FUNCTION F_ROUNDREAL : REAL
VAR_INPUT
	rValue		: REAL; // Input Value
	iDecNumber	: INT; 	// Numbers after decimal point
END_VAR
VAR
	rOutValue	: REAL;
END_VAR

rOutValue := rValue * EXPT(10,iDecNumber);
rOutValue := TRUNC(rOutValue) / EXPT(10,iDecNumber);
F_ROUNDREAL := rOutValue;

END_FUNCTION

(* stored: Version 1.1.0.1, ProductVersion 3.1.4024.9
   POU F_ROUNDREAL: Id {fe6e4e1f-2305-4c5c-9f1d-a0c02cbd7da5}, SpecialFunc None *)
